(* IEC 61131-3 sources: SIGMATEK-Jumag-Utils-Examples/dateTime/Class/dateTimeComponents, 1 file *)

(* ---- dateTimeComponents.st ---- *)
(*!
<Class
	Name               = "dateTimeComponents"
	Revision           = "0.0"
	RealtimeTask       = "false"
	CyclicTask         = "true"
	DefCyclictime      = "100 ms"
	BackgroundTask     = "false"
	Sigmatek           = "false"
	OSInterface        = "false"
	HighPriority       = "false"
	Automatic          = "false"
	UpdateMode         = "Prescan"
	SharedCommandTable = "true"
	Objectsize         = "(284,120)">
	<Channels>
		<Server Name="ClassSvr" Visualized="false" Initialize="false" WriteProtected="true" Retentive="false"/>
		<Server Name="Day" Visualized="false" Initialize="false" WriteProtected="true" Retentive="false"/>
		<Server Name="Hour" Visualized="false" Initialize="false" WriteProtected="true" Retentive="false"/>
		<Server Name="Minute" Visualized="false" Initialize="false" WriteProtected="true" Retentive="false"/>
		<Server Name="Month" Visualized="false" Initialize="false" WriteProtected="true" Retentive="false"/>
		<Server Name="Second" Visualized="false" Initialize="false" WriteProtected="true" Retentive="false"/>
		<Server Name="Year" Visualized="false" Initialize="false" WriteProtected="true" Retentive="false"/>
		<Client Name="cSysDate" Required="true" Internal="false"/>
		<Client Name="cSysTime" Required="true" Internal="false"/>
	</Channels>
	<Separators>
		<Servers>
			<SepChn Position="4"/>
		</Servers>
	</Separators>
	<Dependencies>
		<Files>
			<File Path=".\Source\getTimeComponents.c"/>
		</Files>
	</Dependencies>
</Class>
*)
dateTimeComponents : CLASS
  //Servers:
	ClassSvr 	: SvrChCmd_DINT;
	Second 	: SvrCh_DINT;
	Minute 	: SvrCh_DINT;
	Hour 	: SvrCh_DINT;
	Day 	: SvrCh_DINT;
	Month 	: SvrCh_DINT;
	Year 	: SvrCh_DINT;
  //Clients:
	cSysDate 	: CltCh_DATE_LSL;
	cSysTime 	: CltCh_TIME_LSL;
  //Variables:
		hd_date 	: HDINT;
		hd_time 	: HDINT;
  //Functions:

	FUNCTION VIRTUAL GLOBAL CyWork
		VAR_INPUT
			EAX 	: UDINT;
		END_VAR
		VAR_OUTPUT
			state (EAX) 	: UDINT;
		END_VAR;
  //Tables:
	FUNCTION @STD
		VAR_OUTPUT
			ret_code	: CONFSTATES;
		END_VAR;
	FUNCTION GLOBAL TAB @CT_;
END_CLASS;

Function Global __cdecl getSecondsFromSysTime
VAR_INPUT
  HEX_SYSTIME : HDINT;
END_VAR
VAR_OUTPUT
  Q : UINT;
END_VAR;

Function Global __cdecl getMinutesFromSysTime
VAR_INPUT
  HEX_SYSTIME : HDINT;
END_VAR
VAR_OUTPUT
  Q : UINT;
END_VAR;

Function Global __cdecl getHoursFromSysTime
VAR_INPUT
  HEX_SYSTIME : HDINT;
END_VAR
VAR_OUTPUT
  Q : UINT;
END_VAR;

Function Global __cdecl getDayFromSysDate
VAR_INPUT
  HEX_SYSDATE : HDINT;
END_VAR
VAR_OUTPUT
  Q : UINT;
END_VAR;

Function Global __cdecl getMonthFromSysDate
VAR_INPUT
  HEX_SYSDATE : HDINT;
END_VAR
VAR_OUTPUT
  Q : UINT;
END_VAR;

Function Global __cdecl getYearFromSysDate
VAR_INPUT
  HEX_SYSDATE : HDINT;
END_VAR
VAR_OUTPUT
  Q : UINT;
END_VAR;

FUNCTION VIRTUAL GLOBAL dateTimeComponents::CyWork
	VAR_INPUT
		EAX 	: UDINT;
	END_VAR
	VAR_OUTPUT
		state (EAX) 	: UDINT;
	END_VAR

  hd_time := cSysTime.Read();
  hd_date := cSysDate.Read();

  Second := getSecondsFromSysTime(HEX_SYSTIME:=hd_time);
  Minute := getMinutesFromSysTime(HEX_SYSTIME:=hd_time);
  Hour  := getHoursFromSysTime(HEX_SYSTIME:=hd_time);

  Day := getDayFromSysDate(HEX_SYSDATE:=hd_date);
  Month := getMonthFromSysDate(HEX_SYSDATE:=hd_date);
  Year := getYearFromSysDate(HEX_SYSDATE:=hd_date);

	state := READY;

END_FUNCTION
